PTP {A1 -92.79630,A2 -57.44470,A3 113.54000,A4 -41.50860,A5 -66.88760,A6 21.46980}
; ---- Setting reference (Base) ----
$BASE = {FRAME: X 0.000,Y 0.000,Z 0.000,A 0.000,B 0.000,C 0.000}
; --------------------------
; ---- Setting tool (TCP) ----
; TOOL_DATA[1] = {FRAME: X 0.000,Y 0.000,Z 10.000,A 0.000,B 0.000,C 0.000}
$TOOL = {FRAME: X 0.000,Y 0.000,Z 10.000,A 0.000,B 0.000,C 0.000}
; $TOOL = TOOL_DATA[1]
; --------------------------
PTP {A1 -82.84020,A2 -58.17100,A3 114.32600,A4 36.64330,A5 -63.73490,A6 -16.65780}
; ---- Setting reference (Base) ----
$BASE = {FRAME: X 0.000,Y 0.000,Z 0.000,A 0.000,B 0.000,C 0.000}
; --------------------------
; ---- Setting tool (TCP) ----
; TOOL_DATA[1] = {FRAME: X 0.000,Y 0.000,Z 10.000,A 0.000,B 0.000,C 0.000}
$TOOL = {FRAME: X 0.000,Y 0.000,Z 10.000,A 0.000,B 0.000,C 0.000}
; $TOOL = TOOL_DATA[1]
; --------------------------
PTP {A1 -87.90140,A2 -58.96310,A3 116.51400,A4 -3.08373,A5 -60.62110,A6 3.10240}
; ---- Setting reference (Base) ----
$BASE = {FRAME: X 0.000,Y 0.000,Z 0.000,A 0.000,B 0.000,C 0.000}
; --------------------------
; ---- Setting tool (TCP) ----
; TOOL_DATA[1] = {FRAME: X 0.000,Y 0.000,Z 10.000,A 0.000,B 0.000,C 0.000}
$TOOL = {FRAME: X 0.000,Y 0.000,Z 10.000,A 0.000,B 0.000,C 0.000}
; $TOOL = TOOL_DATA[1]
; --------------------------
PTP {A1 -87.90140,A2 -58.96310,A3 116.51400,A4 -3.08373,A5 -60.62110,A6 -26.89760}
; ---- Setting reference (Base) ----
$BASE = {FRAME: X 0.000,Y 0.000,Z 0.000,A 0.000,B 0.000,C 0.000}
; --------------------------
; ---- Setting tool (TCP) ----
; TOOL_DATA[1] = {FRAME: X 0.000,Y 0.000,Z 10.000,A 0.000,B 0.000,C 0.000}
$TOOL = {FRAME: X 0.000,Y 0.000,Z 10.000,A 0.000,B 0.000,C 0.000}
; $TOOL = TOOL_DATA[1]
; --------------------------
PTP {A1 -87.90140,A2 -58.96310,A3 116.51400,A4 -3.08373,A5 -60.62110,A6 33.10240}
; ---- Setting reference (Base) ----
$BASE = {FRAME: X 0.000,Y 0.000,Z 0.000,A 0.000,B 0.000,C 0.000}
; --------------------------
; ---- Setting tool (TCP) ----
; TOOL_DATA[1] = {FRAME: X 0.000,Y 0.000,Z 10.000,A 0.000,B 0.000,C 0.000}
$TOOL = {FRAME: X 0.000,Y 0.000,Z 10.000,A 0.000,B 0.000,C 0.000}
; $TOOL = TOOL_DATA[1]
; --------------------------
PTP {A1 -87.90140,A2 -58.96310,A3 116.51400,A4 -3.08373,A5 -60.62110,A6 3.10240}
; ---- Setting reference (Base) ----
$BASE = {FRAME: X 0.000,Y 0.000,Z 0.000,A 0.000,B 0.000,C 0.000}
; --------------------------
; ---- Setting tool (TCP) ----
; TOOL_DATA[1] = {FRAME: X 0.000,Y 0.000,Z 10.000,A 0.000,B 0.000,C 0.000}
$TOOL = {FRAME: X 0.000,Y 0.000,Z 10.000,A 0.000,B 0.000,C 0.000}
; $TOOL = TOOL_DATA[1]
; --------------------------
PTP {A1 -89.11650,A2 -58.86460,A3 116.39800,A4 -4.47580,A5 -60.64680,A6 3.85034}
; ---- Setting reference (Base) ----
$BASE = {FRAME: X 0.000,Y 0.000,Z 0.000,A 0.000,B 0.000,C 0.000}
; --------------------------
; ---- Setting tool (TCP) ----
; TOOL_DATA[1] = {FRAME: X 0.000,Y 0.000,Z 10.000,A 0.000,B 0.000,C 0.000}
$TOOL = {FRAME: X 0.000,Y 0.000,Z 10.000,A 0.000,B 0.000,C 0.000}
; $TOOL = TOOL_DATA[1]
; --------------------------
PTP {A1 -93.96270,A2 -57.26530,A3 113.25300,A4 -42.71090,A5 -67.24510,A6 22.07250}
; ---- Setting reference (Base) ----
$BASE = {FRAME: X 0.000,Y 0.000,Z 0.000,A 0.000,B 0.000,C 0.000}
; --------------------------
; ---- Setting tool (TCP) ----
; TOOL_DATA[1] = {FRAME: X 0.000,Y 0.000,Z 10.000,A 0.000,B 0.000,C 0.000}
$TOOL = {FRAME: X 0.000,Y 0.000,Z 10.000,A 0.000,B 0.000,C 0.000}
; $TOOL = TOOL_DATA[1]
; --------------------------
PTP {A1 -84.03000,A2 -58.15880,A3 114.38500,A4 35.36770,A5 -63.40330,A6 -16.01290}
; ---- Setting reference (Base) ----
$BASE = {FRAME: X 0.000,Y 0.000,Z 0.000,A 0.000,B 0.000,C 0.000}
; --------------------------
; ---- Setting tool (TCP) ----
; TOOL_DATA[1] = {FRAME: X 0.000,Y 0.000,Z 10.000,A 0.000,B 0.000,C 0.000}
$TOOL = {FRAME: X 0.000,Y 0.000,Z 10.000,A 0.000,B 0.000,C 0.000}
; $TOOL = TOOL_DATA[1]
; --------------------------
PTP {A1 -89.11650,A2 -58.86460,A3 116.39800,A4 -4.47580,A5 -60.64680,A6 3.85034}
; ---- Setting reference (Base) ----
$BASE = {FRAME: X 0.000,Y 0.000,Z 0.000,A 0.000,B 0.000,C 0.000}
; --------------------------
; ---- Setting tool (TCP) ----
; TOOL_DATA[1] = {FRAME: X 0.000,Y 0.000,Z 10.000,A 0.000,B 0.000,C 0.000}
$TOOL = {FRAME: X 0.000,Y 0.000,Z 10.000,A 0.000,B 0.000,C 0.000}
; $TOOL = TOOL_DATA[1]
; --------------------------
PTP {A1 -89.11650,A2 -58.86460,A3 116.39800,A4 -4.47580,A5 -60.64680,A6 -26.14970}
; ---- Setting reference (Base) ----
$BASE = {FRAME: X 0.000,Y 0.000,Z 0.000,A 0.000,B 0.000,C 0.000}
; --------------------------
; ---- Setting tool (TCP) ----
; TOOL_DATA[1] = {FRAME: X 0.000,Y 0.000,Z 10.000,A 0.000,B 0.000,C 0.000}
$TOOL = {FRAME: X 0.000,Y 0.000,Z 10.000,A 0.000,B 0.000,C 0.000}
; $TOOL = TOOL_DATA[1]
; --------------------------
PTP {A1 -89.11650,A2 -58.86460,A3 116.39800,A4 -4.47580,A5 -60.64680,A6 33.85030}
; ---- Setting reference (Base) ----
$BASE = {FRAME: X 0.000,Y 0.000,Z 0.000,A 0.000,B 0.000,C 0.000}
; --------------------------
; ---- Setting tool (TCP) ----
; TOOL_DATA[1] = {FRAME: X 0.000,Y 0.000,Z 10.000,A 0.000,B 0.000,C 0.000}
$TOOL = {FRAME: X 0.000,Y 0.000,Z 10.000,A 0.000,B 0.000,C 0.000}
; $TOOL = TOOL_DATA[1]
; --------------------------
PTP {A1 -89.11650,A2 -58.86460,A3 116.39800,A4 -4.47580,A5 -60.64680,A6 3.85034}
; ---- Setting reference (Base) ----
$BASE = {FRAME: X 0.000,Y 0.000,Z 0.000,A 0.000,B 0.000,C 0.000}
; --------------------------
; ---- Setting tool (TCP) ----
; TOOL_DATA[1] = {FRAME: X 0.000,Y 0.000,Z 10.000,A 0.000,B 0.000,C 0.000}
$TOOL = {FRAME: X 0.000,Y 0.000,Z 10.000,A 0.000,B 0.000,C 0.000}
; $TOOL = TOOL_DATA[1]
; --------------------------
PTP {A1 -90.32800,A2 -58.74610,A3 116.24000,A4 -5.86404,A5 -60.66670,A6 4.59780}
; ---- Setting reference (Base) ----
$BASE = {FRAME: X 0.000,Y 0.000,Z 0.000,A 0.000,B 0.000,C 0.000}
; --------------------------
; ---- Setting tool (TCP) ----
; TOOL_DATA[1] = {FRAME: X 0.000,Y 0.000,Z 10.000,A 0.000,B 0.000,C 0.000}
$TOOL = {FRAME: X 0.000,Y 0.000,Z 10.000,A 0.000,B 0.000,C 0.000}
; $TOOL = TOOL_DATA[1]
; --------------------------
PTP {A1 -95.12170,A2 -57.06650,A3 112.92600,A4 -43.90390,A5 -67.59720,A6 22.67950}
; ---- Setting reference (Base) ----
$BASE = {FRAME: X 0.000,Y 0.000,Z 0.000,A 0.000,B 0.000,C 0.000}
; --------------------------
; ---- Setting tool (TCP) ----
; TOOL_DATA[1] = {FRAME: X 0.000,Y 0.000,Z 10.000,A 0.000,B 0.000,C 0.000}
$TOOL = {FRAME: X 0.000,Y 0.000,Z 10.000,A 0.000,B 0.000,C 0.000}
; $TOOL = TOOL_DATA[1]
; --------------------------
PTP {A1 -85.22070,A2 -58.12630,A3 114.40200,A4 34.08900,A5 -63.06770,A6 -15.37200}
; ---- Setting reference (Base) ----
$BASE = {FRAME: X 0.000,Y 0.000,Z 0.000,A 0.000,B 0.000,C 0.000}
; --------------------------
; ---- Setting tool (TCP) ----
; TOOL_DATA[1] = {FRAME: X 0.000,Y 0.000,Z 10.000,A 0.000,B 0.000,C 0.000}
$TOOL = {FRAME: X 0.000,Y 0.000,Z 10.000,A 0.000,B 0.000,C 0.000}
; $TOOL = TOOL_DATA[1]
; --------------------------
PTP {A1 -90.32800,A2 -58.74610,A3 116.24000,A4 -5.86404,A5 -60.66670,A6 4.59780}
; ---- Setting reference (Base) ----
$BASE = {FRAME: X 0.000,Y 0.000,Z 0.000,A 0.000,B 0.000,C 0.000}
; --------------------------
; ---- Setting tool (TCP) ----
; TOOL_DATA[1] = {FRAME: X 0.000,Y 0.000,Z 10.000,A 0.000,B 0.000,C 0.000}
$TOOL = {FRAME: X 0.000,Y 0.000,Z 10.000,A 0.000,B 0.000,C 0.000}
; $TOOL = TOOL_DATA[1]
; --------------------------
PTP {A1 -90.32800,A2 -58.74610,A3 116.24000,A4 -5.86404,A5 -60.66670,A6 -25.40220}
; ---- Setting reference (Base) ----
$BASE = {FRAME: X 0.000,Y 0.000,Z 0.000,A 0.000,B 0.000,C 0.000}
; --------------------------
; ---- Setting tool (TCP) ----
; TOOL_DATA[1] = {FRAME: X 0.000,Y 0.000,Z 10.000,A 0.000,B 0.000,C 0.000}
$TOOL = {FRAME: X 0.000,Y 0.000,Z 10.000,A 0.000,B 0.000,C 0.000}
; $TOOL = TOOL_DATA[1]
; --------------------------
PTP {A1 -90.32800,A2 -58.74610,A3 116.24000,A4 -5.86404,A5 -60.66670,A6 34.59780}
; ---- Setting reference (Base) ----
$BASE = {FRAME: X 0.000,Y 0.000,Z 0.000,A 0.000,B 0.000,C 0.000}
; --------------------------
; ---- Setting tool (TCP) ----
; TOOL_DATA[1] = {FRAME: X 0.000,Y 0.000,Z 10.000,A 0.000,B 0.000,C 0.000}
$TOOL = {FRAME: X 0.000,Y 0.000,Z 10.000,A 0.000,B 0.000,C 0.000}
; $TOOL = TOOL_DATA[1]
; --------------------------
PTP {A1 -90.32800,A2 -58.74610,A3 116.24000,A4 -5.86404,A5 -60.66670,A6 4.59780}
; ---- Setting reference (Base) ----
$BASE = {FRAME: X 0.000,Y 0.000,Z 0.000,A 0.000,B 0.000,C 0.000}
; --------------------------
; ---- Setting tool (TCP) ----
; TOOL_DATA[1] = {FRAME: X 0.000,Y 0.000,Z 10.000,A 0.000,B 0.000,C 0.000}
$TOOL = {FRAME: X 0.000,Y 0.000,Z 10.000,A 0.000,B 0.000,C 0.000}
; $TOOL = TOOL_DATA[1]
; --------------------------
PTP {A1 -91.53490,A2 -58.60780,A3 116.04100,A4 -7.24767,A5 -60.68070,A6 5.34536}
; ---- Setting reference (Base) ----
$BASE = {FRAME: X 0.000,Y 0.000,Z 0.000,A 0.000,B 0.000,C 0.000}
; --------------------------
; ---- Setting tool (TCP) ----
; TOOL_DATA[1] = {FRAME: X 0.000,Y 0.000,Z 10.000,A 0.000,B 0.000,C 0.000}
$TOOL = {FRAME: X 0.000,Y 0.000,Z 10.000,A 0.000,B 0.000,C 0.000}
; $TOOL = TOOL_DATA[1]
; --------------------------
PTP {A1 -96.27250,A2 -56.84850,A3 112.55900,A4 -45.08700,A5 -67.94420,A6 23.29130}
; ---- Setting reference (Base) ----
$BASE = {FRAME: X 0.000,Y 0.000,Z 0.000,A 0.000,B 0.000,C 0.000}
; --------------------------
; ---- Setting tool (TCP) ----
; TOOL_DATA[1] = {FRAME: X 0.000,Y 0.000,Z 10.000,A 0.000,B 0.000,C 0.000}
$TOOL = {FRAME: X 0.000,Y 0.000,Z 10.000,A 0.000,B 0.000,C 0.000}
; $TOOL = TOOL_DATA[1]
; --------------------------
PTP {A1 -86.41140,A2 -58.07360,A3 114.37900,A4 32.80810,A5 -62.72770,A6 -14.73470}
; ---- Setting reference (Base) ----
$BASE = {FRAME: X 0.000,Y 0.000,Z 0.000,A 0.000,B 0.000,C 0.000}
; --------------------------
; ---- Setting tool (TCP) ----
; TOOL_DATA[1] = {FRAME: X 0.000,Y 0.000,Z 10.000,A 0.000,B 0.000,C 0.000}
$TOOL = {FRAME: X 0.000,Y 0.000,Z 10.000,A 0.000,B 0.000,C 0.000}
; $TOOL = TOOL_DATA[1]
; --------------------------
PTP {A1 -91.53490,A2 -58.60780,A3 116.04100,A4 -7.24767,A5 -60.68070,A6 5.34536}
; ---- Setting reference (Base) ----
$BASE = {FRAME: X 0.000,Y 0.000,Z 0.000,A 0.000,B 0.000,C 0.000}
; --------------------------
; ---- Setting tool (TCP) ----
; TOOL_DATA[1] = {FRAME: X 0.000,Y 0.000,Z 10.000,A 0.000,B 0.000,C 0.000}
$TOOL = {FRAME: X 0.000,Y 0.000,Z 10.000,A 0.000,B 0.000,C 0.000}
; $TOOL = TOOL_DATA[1]
; --------------------------
PTP {A1 -91.53490,A2 -58.60780,A3 116.04100,A4 -7.24767,A5 -60.68070,A6 -24.65460}
; ---- Setting reference (Base) ----
$BASE = {FRAME: X 0.000,Y 0.000,Z 0.000,A 0.000,B 0.000,C 0.000}
; --------------------------
; ---- Setting tool (TCP) ----
; TOOL_DATA[1] = {FRAME: X 0.000,Y 0.000,Z 10.000,A 0.000,B 0.000,C 0.000}
$TOOL = {FRAME: X 0.000,Y 0.000,Z 10.000,A 0.000,B 0.000,C 0.000}
; $TOOL = TOOL_DATA[1]
; --------------------------
PTP {A1 -91.53490,A2 -58.60780,A3 116.04100,A4 -7.24767,A5 -60.68070,A6 35.34540}
; ---- Setting reference (Base) ----
$BASE = {FRAME: X 0.000,Y 0.000,Z 0.000,A 0.000,B 0.000,C 0.000}
; --------------------------
; ---- Setting tool (TCP) ----
; TOOL_DATA[1] = {FRAME: X 0.000,Y 0.000,Z 10.000,A 0.000,B 0.000,C 0.000}
$TOOL = {FRAME: X 0.000,Y 0.000,Z 10.000,A 0.000,B 0.000,C 0.000}
; $TOOL = TOOL_DATA[1]
; --------------------------
PTP {A1 -91.53490,A2 -58.60780,A3 116.04100,A4 -7.24767,A5 -60.68070,A6 5.34536}
; ---- Setting reference (Base) ----
$BASE = {FRAME: X 0.000,Y 0.000,Z 0.000,A 0.000,B 0.000,C 0.000}
; --------------------------
; ---- Setting tool (TCP) ----
; TOOL_DATA[1] = {FRAME: X 0.000,Y 0.000,Z 10.000,A 0.000,B 0.000,C 0.000}
$TOOL = {FRAME: X 0.000,Y 0.000,Z 10.000,A 0.000,B 0.000,C 0.000}
; $TOOL = TOOL_DATA[1]
; --------------------------
PTP {A1 -92.73610,A2 -58.44970,A3 115.80100,A4 -8.62593,A5 -60.68870,A6 6.09363}
; ---- Setting reference (Base) ----
$BASE = {FRAME: X 0.000,Y 0.000,Z 0.000,A 0.000,B 0.000,C 0.000}
; --------------------------
; ---- Setting tool (TCP) ----
; TOOL_DATA[1] = {FRAME: X 0.000,Y 0.000,Z 10.000,A 0.000,B 0.000,C 0.000}
$TOOL = {FRAME: X 0.000,Y 0.000,Z 10.000,A 0.000,B 0.000,C 0.000}
; $TOOL = TOOL_DATA[1]
; --------------------------
PTP {A1 -97.41430,A2 -56.61130,A3 112.15100,A4 -46.25940,A5 -68.28620,A6 23.90820}
; ---- Setting reference (Base) ----
$BASE = {FRAME: X 0.000,Y 0.000,Z 0.000,A 0.000,B 0.000,C 0.000}
; --------------------------
; ---- Setting tool (TCP) ----
; TOOL_DATA[1] = {FRAME: X 0.000,Y 0.000,Z 10.000,A 0.000,B 0.000,C 0.000}
$TOOL = {FRAME: X 0.000,Y 0.000,Z 10.000,A 0.000,B 0.000,C 0.000}
; $TOOL = TOOL_DATA[1]
; --------------------------
PTP {A1 -87.60090,A2 -58.00090,A3 114.31400,A4 31.52610,A5 -62.38310,A6 -14.10050}
; ---- Setting reference (Base) ----
$BASE = {FRAME: X 0.000,Y 0.000,Z 0.000,A 0.000,B 0.000,C 0.000}
; --------------------------
; ---- Setting tool (TCP) ----
; TOOL_DATA[1] = {FRAME: X 0.000,Y 0.000,Z 10.000,A 0.000,B 0.000,C 0.000}
$TOOL = {FRAME: X 0.000,Y 0.000,Z 10.000,A 0.000,B 0.000,C 0.000}
; $TOOL = TOOL_DATA[1]
; --------------------------
PTP {A1 -92.73610,A2 -58.44970,A3 115.80100,A4 -8.62593,A5 -60.68870,A6 6.09363}
; ---- Setting reference (Base) ----
$BASE = {FRAME: X 0.000,Y 0.000,Z 0.000,A 0.000,B 0.000,C 0.000}
; --------------------------
; ---- Setting tool (TCP) ----
; TOOL_DATA[1] = {FRAME: X 0.000,Y 0.000,Z 10.000,A 0.000,B 0.000,C 0.000}
$TOOL = {FRAME: X 0.000,Y 0.000,Z 10.000,A 0.000,B 0.000,C 0.000}
; $TOOL = TOOL_DATA[1]
; --------------------------
PTP {A1 -92.73610,A2 -58.44970,A3 115.80100,A4 -8.62593,A5 -60.68870,A6 -23.90640}
; ---- Setting reference (Base) ----
$BASE = {FRAME: X 0.000,Y 0.000,Z 0.000,A 0.000,B 0.000,C 0.000}
; --------------------------
; ---- Setting tool (TCP) ----
; TOOL_DATA[1] = {FRAME: X 0.000,Y 0.000,Z 10.000,A 0.000,B 0.000,C 0.000}
$TOOL = {FRAME: X 0.000,Y 0.000,Z 10.000,A 0.000,B 0.000,C 0.000}
; $TOOL = TOOL_DATA[1]
; --------------------------
PTP {A1 -92.73610,A2 -58.44970,A3 115.80100,A4 -8.62593,A5 -60.68870,A6 36.09360}
; ---- Setting reference (Base) ----
$BASE = {FRAME: X 0.000,Y 0.000,Z 0.000,A 0.000,B 0.000,C 0.000}
; --------------------------
; ---- Setting tool (TCP) ----
; TOOL_DATA[1] = {FRAME: X 0.000,Y 0.000,Z 10.000,A 0.000,B 0.000,C 0.000}
$TOOL = {FRAME: X 0.000,Y 0.000,Z 10.000,A 0.000,B 0.000,C 0.000}
; $TOOL = TOOL_DATA[1]
; --------------------------
PTP {A1 -92.73610,A2 -58.44970,A3 115.80100,A4 -8.62593,A5 -60.68870,A6 6.09363}
; ---- Setting reference (Base) ----
$BASE = {FRAME: X 0.000,Y 0.000,Z 0.000,A 0.000,B 0.000,C 0.000}
; --------------------------
; ---- Setting tool (TCP) ----
; TOOL_DATA[1] = {FRAME: X 0.000,Y 0.000,Z 10.000,A 0.000,B 0.000,C 0.000}
$TOOL = {FRAME: X 0.000,Y 0.000,Z 10.000,A 0.000,B 0.000,C 0.000}
; $TOOL = TOOL_DATA[1]
; --------------------------
PTP {A1 -93.93060,A2 -58.27190,A3 115.52000,A4 -9.99809,A5 -60.69060,A6 6.84322}
; ---- Setting reference (Base) ----
$BASE = {FRAME: X 0.000,Y 0.000,Z 0.000,A 0.000,B 0.000,C 0.000}
; --------------------------
; ---- Setting tool (TCP) ----
; TOOL_DATA[1] = {FRAME: X 0.000,Y 0.000,Z 10.000,A 0.000,B 0.000,C 0.000}
$TOOL = {FRAME: X 0.000,Y 0.000,Z 10.000,A 0.000,B 0.000,C 0.000}
; $TOOL = TOOL_DATA[1]
; --------------------------
PTP {A1 -98.54630,A2 -56.35520,A3 111.70400,A4 -47.42020,A5 -68.62350,A6 24.53060}
; ---- Setting reference (Base) ----
$BASE = {FRAME: X 0.000,Y 0.000,Z 0.000,A 0.000,B 0.000,C 0.000}
; --------------------------
; ---- Setting tool (TCP) ----
; TOOL_DATA[1] = {FRAME: X 0.000,Y 0.000,Z 10.000,A 0.000,B 0.000,C 0.000}
$TOOL = {FRAME: X 0.000,Y 0.000,Z 10.000,A 0.000,B 0.000,C 0.000}
; $TOOL = TOOL_DATA[1]
; --------------------------
PTP {A1 -88.78840,A2 -57.90820,A3 114.20800,A4 30.24370,A5 -62.03350,A6 -13.46930}
; ---- Setting reference (Base) ----
$BASE = {FRAME: X 0.000,Y 0.000,Z 0.000,A 0.000,B 0.000,C 0.000}
; --------------------------
; ---- Setting tool (TCP) ----
; TOOL_DATA[1] = {FRAME: X 0.000,Y 0.000,Z 10.000,A 0.000,B 0.000,C 0.000}
$TOOL = {FRAME: X 0.000,Y 0.000,Z 10.000,A 0.000,B 0.000,C 0.000}
; $TOOL = TOOL_DATA[1]
; --------------------------
PTP {A1 -93.93060,A2 -58.27190,A3 115.52000,A4 -9.99809,A5 -60.69060,A6 6.84322}
; ---- Setting reference (Base) ----
$BASE = {FRAME: X 0.000,Y 0.000,Z 0.000,A 0.000,B 0.000,C 0.000}
; --------------------------
; ---- Setting tool (TCP) ----
; TOOL_DATA[1] = {FRAME: X 0.000,Y 0.000,Z 10.000,A 0.000,B 0.000,C 0.000}
$TOOL = {FRAME: X 0.000,Y 0.000,Z 10.000,A 0.000,B 0.000,C 0.000}
; $TOOL = TOOL_DATA[1]
; --------------------------
PTP {A1 -93.93060,A2 -58.27190,A3 115.52000,A4 -9.99809,A5 -60.69060,A6 -23.15680}
; ---- Setting reference (Base) ----
$BASE = {FRAME: X 0.000,Y 0.000,Z 0.000,A 0.000,B 0.000,C 0.000}
; --------------------------
; ---- Setting tool (TCP) ----
; TOOL_DATA[1] = {FRAME: X 0.000,Y 0.000,Z 10.000,A 0.000,B 0.000,C 0.000}
$TOOL = {FRAME: X 0.000,Y 0.000,Z 10.000,A 0.000,B 0.000,C 0.000}
; $TOOL = TOOL_DATA[1]
; --------------------------
PTP {A1 -93.93060,A2 -58.27190,A3 115.52000,A4 -9.99809,A5 -60.69060,A6 36.84320}
; ---- Setting reference (Base) ----
$BASE = {FRAME: X 0.000,Y 0.000,Z 0.000,A 0.000,B 0.000,C 0.000}
; --------------------------
; ---- Setting tool (TCP) ----
; TOOL_DATA[1] = {FRAME: X 0.000,Y 0.000,Z 10.000,A 0.000,B 0.000,C 0.000}
$TOOL = {FRAME: X 0.000,Y 0.000,Z 10.000,A 0.000,B 0.000,C 0.000}
; $TOOL = TOOL_DATA[1]
; --------------------------
PTP {A1 -93.93060,A2 -58.27190,A3 115.52000,A4 -9.99809,A5 -60.69060,A6 6.84322}
; ---- Setting reference (Base) ----
$BASE = {FRAME: X 0.000,Y 0.000,Z 0.000,A 0.000,B 0.000,C 0.000}
; --------------------------
; ---- Setting tool (TCP) ----
; TOOL_DATA[1] = {FRAME: X 0.000,Y 0.000,Z 10.000,A 0.000,B 0.000,C 0.000}
$TOOL = {FRAME: X 0.000,Y 0.000,Z 10.000,A 0.000,B 0.000,C 0.000}
; $TOOL = TOOL_DATA[1]
; --------------------------
PTP {A1 -95.11750,A2 -58.07480,A3 115.19700,A4 -11.36350,A5 -60.68670,A6 7.59471}
; ---- Setting reference (Base) ----
$BASE = {FRAME: X 0.000,Y 0.000,Z 0.000,A 0.000,B 0.000,C 0.000}
; --------------------------
; ---- Setting tool (TCP) ----
; TOOL_DATA[1] = {FRAME: X 0.000,Y 0.000,Z 10.000,A 0.000,B 0.000,C 0.000}
$TOOL = {FRAME: X 0.000,Y 0.000,Z 10.000,A 0.000,B 0.000,C 0.000}
; $TOOL = TOOL_DATA[1]
; --------------------------
PTP {A1 -99.66770,A2 -56.08030,A3 111.21600,A4 -48.56890,A5 -68.95630,A6 25.15890}
; ---- Setting reference (Base) ----
$BASE = {FRAME: X 0.000,Y 0.000,Z 0.000,A 0.000,B 0.000,C 0.000}
; --------------------------
; ---- Setting tool (TCP) ----
; TOOL_DATA[1] = {FRAME: X 0.000,Y 0.000,Z 10.000,A 0.000,B 0.000,C 0.000}
$TOOL = {FRAME: X 0.000,Y 0.000,Z 10.000,A 0.000,B 0.000,C 0.000}
; $TOOL = TOOL_DATA[1]
; --------------------------
PTP {A1 -89.97270,A2 -57.79550,A3 114.06100,A4 28.96200,A5 -61.67860,A6 -12.84040}
; ---- Setting reference (Base) ----
$BASE = {FRAME: X 0.000,Y 0.000,Z 0.000,A 0.000,B 0.000,C 0.000}
; --------------------------
; ---- Setting tool (TCP) ----
; TOOL_DATA[1] = {FRAME: X 0.000,Y 0.000,Z 10.000,A 0.000,B 0.000,C 0.000}
$TOOL = {FRAME: X 0.000,Y 0.000,Z 10.000,A 0.000,B 0.000,C 0.000}
; $TOOL = TOOL_DATA[1]
; --------------------------
PTP {A1 -95.11750,A2 -58.07480,A3 115.19700,A4 -11.36350,A5 -60.68670,A6 7.59471}
; ---- Setting reference (Base) ----
$BASE = {FRAME: X 0.000,Y 0.000,Z 0.000,A 0.000,B 0.000,C 0.000}
; --------------------------
; ---- Setting tool (TCP) ----
; TOOL_DATA[1] = {FRAME: X 0.000,Y 0.000,Z 10.000,A 0.000,B 0.000,C 0.000}
$TOOL = {FRAME: X 0.000,Y 0.000,Z 10.000,A 0.000,B 0.000,C 0.000}
; $TOOL = TOOL_DATA[1]
; --------------------------
PTP {A1 -95.11750,A2 -58.07480,A3 115.19700,A4 -11.36350,A5 -60.68670,A6 -22.40530}
; ---- Setting reference (Base) ----
$BASE = {FRAME: X 0.000,Y 0.000,Z 0.000,A 0.000,B 0.000,C 0.000}
; --------------------------
; ---- Setting tool (TCP) ----
; TOOL_DATA[1] = {FRAME: X 0.000,Y 0.000,Z 10.000,A 0.000,B 0.000,C 0.000}
$TOOL = {FRAME: X 0.000,Y 0.000,Z 10.000,A 0.000,B 0.000,C 0.000}
; $TOOL = TOOL_DATA[1]
; --------------------------
PTP {A1 -95.11750,A2 -58.07480,A3 115.19700,A4 -11.36350,A5 -60.68670,A6 37.59470}
; ---- Setting reference (Base) ----
$BASE = {FRAME: X 0.000,Y 0.000,Z 0.000,A 0.000,B 0.000,C 0.000}
; --------------------------
; ---- Setting tool (TCP) ----
; TOOL_DATA[1] = {FRAME: X 0.000,Y 0.000,Z 10.000,A 0.000,B 0.000,C 0.000}
$TOOL = {FRAME: X 0.000,Y 0.000,Z 10.000,A 0.000,B 0.000,C 0.000}
; $TOOL = TOOL_DATA[1]
; --------------------------
PTP {A1 -95.11750,A2 -58.07480,A3 115.19700,A4 -11.36350,A5 -60.68670,A6 7.59471}
; ---- Setting reference (Base) ----
$BASE = {FRAME: X 0.000,Y 0.000,Z 0.000,A 0.000,B 0.000,C 0.000}
; --------------------------
; ---- Setting tool (TCP) ----
; TOOL_DATA[1] = {FRAME: X 0.000,Y 0.000,Z 10.000,A 0.000,B 0.000,C 0.000}
$TOOL = {FRAME: X 0.000,Y 0.000,Z 10.000,A 0.000,B 0.000,C 0.000}
; $TOOL = TOOL_DATA[1]
; --------------------------
PTP {A1 -96.29580,A2 -57.85820,A3 114.83400,A4 -12.72140,A5 -60.67670,A6 8.34871}
; ---- Setting reference (Base) ----
$BASE = {FRAME: X 0.000,Y 0.000,Z 0.000,A 0.000,B 0.000,C 0.000}
; --------------------------
; ---- Setting tool (TCP) ----
; TOOL_DATA[1] = {FRAME: X 0.000,Y 0.000,Z 10.000,A 0.000,B 0.000,C 0.000}
$TOOL = {FRAME: X 0.000,Y 0.000,Z 10.000,A 0.000,B 0.000,C 0.000}
; $TOOL = TOOL_DATA[1]
; --------------------------
PTP {A1 -100.77800,A2 -55.78670,A3 110.68900,A4 -49.70460,A5 -69.28490,A6 25.79350}
; ---- Setting reference (Base) ----
$BASE = {FRAME: X 0.000,Y 0.000,Z 0.000,A 0.000,B 0.000,C 0.000}
; --------------------------
; ---- Setting tool (TCP) ----

; Continue running program as cascaded execution
Kuka_Relative_Mo2()

END
